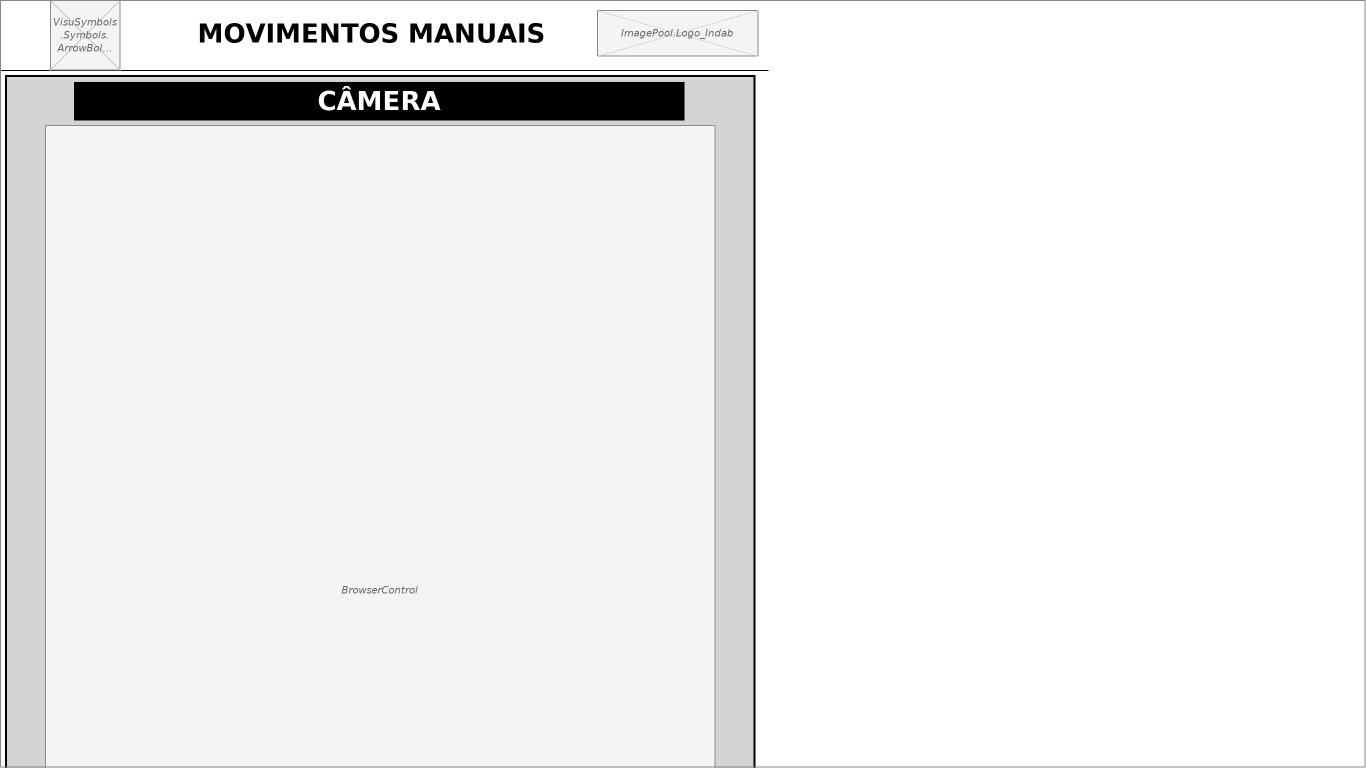
VISUALIZATION Tela_Manual_3  // 1366x768
    Line (0,70) (768,70)
    Line (0,1312) (768,1312)
    Image (597,10 161x46), image: ImagePool.Logo_Indab
    Rectangle (584,1340 180x24), "%t[dd/MM/yyyy]"
    Rectangle (584,1316 180x24), "%t[HH:mm:ss]"
    Label (153,7 437x53), "MOVIMENTOS MANUAIS"
    Button (15,1315 175x45), "RECEITAS"
        OnMouseClick: change screen: Tela_Receita
    Button (375,1315 175x45), "MANUTENÇÃO"
        OnMouseClick: change screen: Tela_Manutencao
    RoundedRectangle (5,75 750x1230)
    Rectangle (74,82 610x38), "CÂMERA", text variable: Recipe_name_Select
    Image (50,0 70x70), image: VisuSymbols.Symbols.ArrowBoldLeft
        OnMouseClick: change screen: Tela_Manual_2
    BrowserControl (45,125 670x930)
        p3734058945: MAIN.sUrlAddressCamera
    Button (195,1315 175x45), "PRODUÇÃO"
        OnMouseClick: change screen: Tela_Producao
    RoundedRectangle (207,1180 150x30), "TRIGGER", input disabled if: NOT MaquinaModoManual
        tap IhmBt_Camera_Trigger
    Rectangle (226,1110 130x25), "ID: %d", text variable: IhmEscr_Camera_SetJob
        OnMouseClick: write the text variable via Default, min 0, max 300
    Rectangle (50,1113 155x20), "Selecionar Job (Job ID):", input disabled if: NOT MaquinaModoManual
    Rectangle (226,1140 130x25), "%.2f s", text variable: IhmEscr_Camera_DelayError
        OnMouseClick: write the text variable via Default, min 0, max 300
    Rectangle (50,1143 130x20), "Delay (ERROR):", input disabled if: NOT MaquinaModoManual
    Rectangle (447,1115 180x22), "Executando Job (Job ID):", input disabled if: NOT MaquinaModoManual
    Rectangle (500,1070 180x27), "Status Câmera", text variable: Recipe_name_Select, input disabled if: NOT MaquinaModoManual
    Rectangle (623,1115 90x22), "%d", text variable: IhmLeit_Camera_JobID, input disabled if: NOT MaquinaModoManual
    Rectangle (109,1070 188x27), "Controle Manual:", text variable: Recipe_name_Select, input disabled if: NOT MaquinaModoManual
    Button (260,1235 240x60), "MODO: %s", text variable: IhmBt_ManualAuto_Text, colour toggle: IhmBt_ManualAuto_Color
        toggle IhmBt_ManualAuto
    RoundedRectangle (50,1180 150x30), "CHANGE JOG", input disabled if: NOT MaquinaModoManual
        tap IhmBt_Camera_ChangeJob
    Rectangle (619,1181 100x30), "%s", colour toggle: IhmLed_Camera_JobResult, input disabled if: NOT MaquinaModoManual
    Lamp1 (653,1146 30x30), variable: IhmLed_Camera_JobCompleted, style: Lamp-Lamp1-Red
    Rectangle (447,1150 180x22), "Job Completed:", input disabled if: NOT MaquinaModoManual
    Rectangle (447,1185 180x22), "Job Result:", input disabled if: NOT MaquinaModoManual
END_VISUALIZATION

(* stored: Version 1.1.0.1, ProductVersion 3.1.4024.11
   Visu Tela_Manual_3: Id {611e0859-6569-4a6f-a753-c415c39f8df9} *)
